(* IEC 61131-3 sources: AXOpen/src/components.rexroth.drives/app/src/IO, 9 files *)

(* ---- HwIdentifiers.st ---- *)
NAMESPACE AXOpen.Components.Rexroth.Drives
    TYPE
        HwIdentifiers : WORD
        (
            ST3_indradrive_HwID :=	WORD#258,
            ST3_indradrive_F_Modul_not_used_ID_FMod_NotUsed_HwID :=	WORD#266,
            ST3_indradrive_Input_9_Words_ID_InMod_9Words_HwID :=	WORD#264,
            ST3_indradrive_Output_13_Words_ID_OutMod_13Words_HwID :=	WORD#263,
            ST3_indradrive_ParamCh_5Words_ID_PaCh_5Words_HwID :=	WORD#265,
            ST3_indradrive_Rack_HwID :=	WORD#261,
            ST3_indradrive_ST3_indradrive_HwID :=	WORD#262,
            ST3_indradrive_ST3_indradrive_DAP_1_HwID :=	WORD#267,
            ST3_indradrive_ST3_indradrive_profinet_HwID :=	WORD#257,
            ST3_indradrive_ST3_indradrive_profinet_Port_1_HwID :=	WORD#259,
            ST3_indradrive_ST3_indradrive_profinet_Port_2_HwID :=	WORD#260,
            plc_line_HwID :=	WORD#32,
            plc_line_Rail_0_HwID :=	WORD#268,
            plc_line_plc_line_HwID :=	WORD#48,
            plc_line_plc_line_CPU_display_1_HwID :=	WORD#54,
            plc_line_plc_line_Card_reader_writer_1_HwID :=	WORD#51,
            plc_line_plc_line_DP_interface_1_HwID :=	WORD#60,
            plc_line_plc_line_OPC_UA_1_HwID :=	WORD#117,
            plc_line_plc_line_profinet_x1_HwID :=	WORD#64,
            plc_line_plc_line_profinet_x1_Port_1_HwID :=	WORD#65,
            plc_line_plc_line_profinet_x1_Port_2_HwID :=	WORD#66,
            plc_line_plc_line_profinet_x2_HwID :=	WORD#72,
            plc_line_plc_line_profinet_x2_Port_3_HwID :=	WORD#73,
            plc_line_plc_line_virtual_communication_interface_HwID :=	WORD#135,
            profinet_plc_line_HwID :=	WORD#256,

            NONE := WORD#0
        );
    END_TYPE
END_NAMESPACE

(* ---- HwInputs.st ---- *)
TYPE
	{S7.extern=ReadWrite}
	HwInputs : STRUCT
		ST3_indradrive_ParamCh_IDN_1 AT %B10 : ARRAY[0..9] OF BYTE;
		ST3_indradrive_Input_9_Words_1 AT %B20 : ARRAY[0..17] OF BYTE;
	END_STRUCT;
END_TYPE

(* ---- HwOutputs.st ---- *)
TYPE
	HwOutputs : STRUCT
		ST3_indradrive_ParamCh_IDN_1 AT %B10 : ARRAY[0..9] OF BYTE;
		ST3_indradrive_Output_13_Words_1 AT %B20 : ARRAY[0..25] OF BYTE;
	END_STRUCT;
END_TYPE

(* ---- Inputs.st ---- *)
NAMESPACE AXOpen.Components.Rexroth.Drives
    TYPE
        {S7.extern=ReadWrite}
        {#ix-attr:[Container(Layout.Wrap)]}
        Inputs : STRUCT
            AxoCtrlxDriveXsc_Inputs_Submodule_1 AT %B0:  WORD;
            AxoCtrlxDriveXsc_Inputs_Submodule_2 AT %B20:  WORD;
            AxoCtrlxDriveXsc_Inputs_Submodule_3 AT %B18:  WORD;
            AxoCtrlxDriveXsc_Inputs_Submodule_4 AT %B2:  WORD;
            AxoCtrlxDriveXsc_Inputs_Submodule_5 AT %B4:  DWORD;
            AxoCtrlxDriveXsc_Inputs_Submodule_6 AT %B12:  DWORD;
            AxoCtrlxDriveXsc_Inputs_Submodule_7 AT %B8:  DWORD;
            AxoCtrlxDriveXsc_Inputs_Submodule_8 AT %B16:  WORD;
            ST3_indradrive_Input_9_Words_0 AT %B24:  WORD;
            ST3_indradrive_Input_9_Words_1 AT %B26:  WORD;
            ST3_indradrive_Input_9_Words_2 AT %B28:  WORD;
            ST3_indradrive_Input_9_Words_3 AT %B30:  WORD;
            ST3_indradrive_Input_9_Words_4 AT %B32:  WORD;
            ST3_indradrive_Input_9_Words_5 AT %B34:  WORD;
            ST3_indradrive_Input_9_Words_6 AT %B36:  WORD;
            ST3_indradrive_Input_9_Words_7 AT %B38:  WORD;
            ST3_indradrive_Input_9_Words_8 AT %B40:  WORD;
            ST3_indradrive_ParamCh_5Words_0 AT %B42:  WORD;
            ST3_indradrive_ParamCh_5Words_1 AT %B44:  WORD;
            ST3_indradrive_ParamCh_5Words_2 AT %B46:  WORD;
            ST3_indradrive_ParamCh_5Words_3 AT %B48:  WORD;
            ST3_indradrive_ParamCh_5Words_4 AT %B50:  WORD;
        END_STRUCT;
    END_TYPE
END_NAMESPACE

(* ---- IoStructures.st ---- *)
NAMESPACE AXOpen.Components.Rexroth.Drives
	TYPE
        {S7.extern=ReadWrite}
        {#ix-attr:[Container(Layout.Wrap)]}
	    AxoCtrlxDriveXsc_Inputs_P_0_0106_0_0__STO_function__Operating_status_Input_Layout : STRUCT
	        Signals_0 AT %B0 : WORD;
	    END_STRUCT;
	END_TYPE

	TYPE
        {S7.extern=ReadWrite}
        {#ix-attr:[Container(Layout.Wrap)]}
	    AxoCtrlxDriveXsc_Inputs_S_0_0084_0_0__Torque_force_feedback_value_Input_Layout : STRUCT
	        Signals_0 AT %B0 : INT;
	    END_STRUCT;
	END_TYPE

	TYPE
        {S7.extern=ReadWrite}
        {#ix-attr:[Container(Layout.Wrap)]}
	    AxoCtrlxDriveXsc_Inputs_S_0_0135_0_0__Drive_status_word__Value_Input_Layout : STRUCT
	        Signals_0 AT %X0.3 : BOOL;
	        Signals_1 AT %X0.4 : BOOL;
	        Signals_2 AT %X0.5 : BOOL;
	        Signals_3 AT %X0.7 : BOOL;
	        Signals_4 AT %X1.0 : BOOL;
	        Signals_5 AT %X1.1 : BOOL;
	        Signals_6 AT %X1.2 : BOOL;
	        Signals_7 AT %X1.4 : BOOL;
	        Signals_8 AT %X1.5 : BOOL;
	        Signals_9 AT %X1.6 : BOOL;
	        Signals_10 AT %X1.7 : BOOL;
	    END_STRUCT;
	END_TYPE

	TYPE
        {S7.extern=ReadWrite}
        {#ix-attr:[Container(Layout.Wrap)]}
	    AxoCtrlxDriveXsc_Inputs_S_0_0144_0_0__Signal_status_word__Value_Input_Layout : STRUCT
	        Signals_0 AT %B0 : WORD;
	    END_STRUCT;
	END_TYPE

	TYPE
        {S7.extern=ReadWrite}
        {#ix-attr:[Container(Layout.Wrap)]}
	    AxoCtrlxDriveXsc_Inputs_S_0_0386_0_0__Position_controller__Position_actual_value_Input_Layout : STRUCT
	        Signals_0 AT %B0 : DINT;
	    END_STRUCT;
	END_TYPE

	TYPE
        {S7.extern=ReadWrite}
        {#ix-attr:[Container(Layout.Wrap)]}
	    AxoCtrlxDriveXsc_Inputs_S_0_0390_0_0__Diagnostic_message__Manufacturer_status_register_Input_Layout : STRUCT
	        Signals_0 AT %B0 : DWORD;
	    END_STRUCT;
	END_TYPE

	TYPE
        {S7.extern=ReadWrite}
        {#ix-attr:[Container(Layout.Wrap)]}
	    AxoCtrlxDriveXsc_Inputs_S_0_0535_0_0__Velocity_controller__Velocity_actual_value_Input_Layout : STRUCT
	        Signals_0 AT %B0 : DINT;
	    END_STRUCT;
	END_TYPE

	TYPE
        {S7.extern=ReadWrite}
        {#ix-attr:[Container(Layout.Wrap)]}
	    AxoCtrlxDriveXsc_Inputs_S_0_1720_0_2__Power_supply_control__Status_word_Input_Layout : STRUCT
	        Signals_0 AT %B0 : WORD;
	    END_STRUCT;
	END_TYPE

	TYPE
        {S7.extern=ReadWrite}
        {#ix-attr:[Container(Layout.Wrap)]}
	    AxoCtrlxDriveXsc_Outputs_S_0_0080_0_0__Torque_force_command_value_Output_Layout : STRUCT
	        Signals_0 AT %B0 : INT;
	    END_STRUCT;
	END_TYPE

	TYPE
        {S7.extern=ReadWrite}
        {#ix-attr:[Container(Layout.Wrap)]}
	    AxoCtrlxDriveXsc_Outputs_S_0_0092_0_0__Torque_force_limitation__Limit_value_bipolar_Output_Layout : STRUCT
	        Signals_0 AT %B0 : WORD;
	    END_STRUCT;
	END_TYPE

	TYPE
        {S7.extern=ReadWrite}
        {#ix-attr:[Container(Layout.Wrap)]}
	    AxoCtrlxDriveXsc_Outputs_S_0_0134_0_0__Master_control_word__Value_Output_Layout : STRUCT
	        Signals_0 AT %X1.0 : BOOL;
	        Signals_1 AT %X1.1 : BOOL;
	        Signals_2 AT %X1.2 : BOOL;
	        Signals_3 AT %X1.5 : BOOL;
	        Signals_4 AT %X1.6 : BOOL;
	        Signals_5 AT %X1.7 : BOOL;
	    END_STRUCT;
	END_TYPE

	TYPE
        {S7.extern=ReadWrite}
        {#ix-attr:[Container(Layout.Wrap)]}
	    AxoCtrlxDriveXsc_Outputs_S_0_0145_0_0__Signal_control_word__Value_Output_Layout : STRUCT
	        Signals_0 AT %B0 : WORD;
	    END_STRUCT;
	END_TYPE

	TYPE
        {S7.extern=ReadWrite}
        {#ix-attr:[Container(Layout.Wrap)]}
	    AxoCtrlxDriveXsc_Outputs_S_0_0193_0_0__Positioning_jerk_Output_Layout : STRUCT
	        Signals_0 AT %B0 : DINT;
	    END_STRUCT;
	END_TYPE

	TYPE
        {S7.extern=ReadWrite}
        {#ix-attr:[Container(Layout.Wrap)]}
	    AxoCtrlxDriveXsc_Outputs_S_0_0259_0_0__Positioning_profile__Profile_velocity_Output_Layout : STRUCT
	        Signals_0 AT %B0 : DWORD;
	    END_STRUCT;
	END_TYPE

	TYPE
        {S7.extern=ReadWrite}
        {#ix-attr:[Container(Layout.Wrap)]}
	    AxoCtrlxDriveXsc_Outputs_S_0_0260_0_0__Positioning_profile__Acceleration_Output_Layout : STRUCT
	        Signals_0 AT %B0 : DINT;
	    END_STRUCT;
	END_TYPE

	TYPE
        {S7.extern=ReadWrite}
        {#ix-attr:[Container(Layout.Wrap)]}
	    AxoCtrlxDriveXsc_Outputs_S_0_0282_0_0__Drive_controlled_positioning__Command_value_Output_Layout : STRUCT
	        Signals_0 AT %B0 : DINT;
	    END_STRUCT;
	END_TYPE

	TYPE
        {S7.extern=ReadWrite}
        {#ix-attr:[Container(Layout.Wrap)]}
	    AxoCtrlxDriveXsc_Outputs_S_0_0359_0_0__Positioning_profile__Deceleration_Output_Layout : STRUCT
	        Signals_0 AT %B0 : DINT;
	    END_STRUCT;
	END_TYPE

	TYPE
        {S7.extern=ReadWrite}
        {#ix-attr:[Container(Layout.Wrap)]}
	    AxoCtrlxDriveXsc_Outputs_S_0_1720_0_1__Power_supply_control__Control_word_Output_Layout : STRUCT
	        Signals_0 AT %B0 : WORD;
	    END_STRUCT;
	END_TYPE

	TYPE
        {S7.extern=ReadWrite}
        {#ix-attr:[Container(Layout.Wrap)]}
	    ST3_indradrive_Input_9_Words_Input_Layout : STRUCT
	        Signals_0 AT %B0 : WORD;
	        Signals_1 AT %B2 : WORD;
	        Signals_2 AT %B4 : WORD;
	        Signals_3 AT %B6 : WORD;
	        Signals_4 AT %B8 : WORD;
	        Signals_5 AT %B10 : WORD;
	        Signals_6 AT %B12 : WORD;
	        Signals_7 AT %B14 : WORD;
	        Signals_8 AT %B16 : WORD;
	    END_STRUCT;
	END_TYPE

	TYPE
        {S7.extern=ReadWrite}
        {#ix-attr:[Container(Layout.Wrap)]}
	    ST3_indradrive_Output_13_Words_Output_Layout : STRUCT
	        Signals_0 AT %B0 : WORD;
	        Signals_1 AT %B2 : WORD;
	        Signals_2 AT %B4 : WORD;
	        Signals_3 AT %B6 : WORD;
	        Signals_4 AT %B8 : WORD;
	        Signals_5 AT %B10 : WORD;
	        Signals_6 AT %B12 : WORD;
	        Signals_7 AT %B14 : WORD;
	        Signals_8 AT %B16 : WORD;
	        Signals_9 AT %B18 : WORD;
	        Signals_10 AT %B20 : WORD;
	        Signals_11 AT %B22 : WORD;
	        Signals_12 AT %B24 : WORD;
	    END_STRUCT;
	END_TYPE

	TYPE
        {S7.extern=ReadWrite}
        {#ix-attr:[Container(Layout.Wrap)]}
	    ST3_indradrive_ParamCh_5Words_Input_Layout : STRUCT
	        Signals_0 AT %B0 : WORD;
	        Signals_1 AT %B2 : WORD;
	        Signals_2 AT %B4 : WORD;
	        Signals_3 AT %B6 : WORD;
	        Signals_4 AT %B8 : WORD;
	    END_STRUCT;
	END_TYPE

	TYPE
        {S7.extern=ReadWrite}
        {#ix-attr:[Container(Layout.Wrap)]}
	    ST3_indradrive_ParamCh_5Words_Output_Layout : STRUCT
	        Signals_5 AT %B0 : WORD;
	        Signals_6 AT %B2 : WORD;
	        Signals_7 AT %B4 : WORD;
	        Signals_8 AT %B6 : WORD;
	        Signals_9 AT %B8 : WORD;
	    END_STRUCT;
	END_TYPE
END_NAMESPACE

(* ---- Outputs.st ---- *)
NAMESPACE AXOpen.Components.Rexroth.Drives
    TYPE
        {S7.extern=ReadWrite}
        {#ix-attr:[Container(Layout.Wrap)]}
        Outputs : STRUCT
	        // Module rexroth_ctrlx_drive/Outputs
	        rexroth_ctrlx_drive_Outputs_S_0_0080_0_0__Torque_force_command_value_Output AT %B24 : rexroth_ctrlx_drive_Outputs_S_0_0080_0_0__Torque_force_command_value_Output_Layout;

	        rexroth_ctrlx_drive_Outputs_S_0_0092_0_0__Torque_force_limitation__Limit_value_bipolar_Output AT %B22 : rexroth_ctrlx_drive_Outputs_S_0_0092_0_0__Torque_force_limitation__Limit_value_bipolar_Output_Layout;

	        rexroth_ctrlx_drive_Outputs_S_0_0134_0_0__Master_control_word__Value_Output AT %B0 : rexroth_ctrlx_drive_Outputs_S_0_0134_0_0__Master_control_word__Value_Output_Layout;

	        rexroth_ctrlx_drive_Outputs_S_0_0145_0_0__Signal_control_word__Value_Output AT %B18 : rexroth_ctrlx_drive_Outputs_S_0_0145_0_0__Signal_control_word__Value_Output_Layout;

	        rexroth_ctrlx_drive_Outputs_S_0_0193_0_0__Positioning_jerk_Output AT %B26 : rexroth_ctrlx_drive_Outputs_S_0_0193_0_0__Positioning_jerk_Output_Layout;

	        rexroth_ctrlx_drive_Outputs_S_0_0259_0_0__Positioning_profile__Profile_velocity_Output AT %B14 : rexroth_ctrlx_drive_Outputs_S_0_0259_0_0__Positioning_profile__Profile_velocity_Output_Layout;

	        rexroth_ctrlx_drive_Outputs_S_0_0260_0_0__Positioning_profile__Acceleration_Output AT %B2 : rexroth_ctrlx_drive_Outputs_S_0_0260_0_0__Positioning_profile__Acceleration_Output_Layout;

	        rexroth_ctrlx_drive_Outputs_S_0_0282_0_0__Drive_controlled_positioning__Command_value_Output AT %B6 : rexroth_ctrlx_drive_Outputs_S_0_0282_0_0__Drive_controlled_positioning__Command_value_Output_Layout;

	        rexroth_ctrlx_drive_Outputs_S_0_0359_0_0__Positioning_profile__Deceleration_Output AT %B10 : rexroth_ctrlx_drive_Outputs_S_0_0359_0_0__Positioning_profile__Deceleration_Output_Layout;

	        rexroth_ctrlx_drive_Outputs_S_0_1720_0_1__Power_supply_control__Control_word_Output AT %B20 : rexroth_ctrlx_drive_Outputs_S_0_1720_0_1__Power_supply_control__Control_word_Output_Layout;

	        // Module rexroth_indradrive/Output_13_Words
	        rexroth_indradrive_Output_13_Words_Output AT %B30 : rexroth_indradrive_Output_13_Words_Output_Layout;

	        rexroth_indradrive_ParamCh_5Words_Output AT %B56 : rexroth_indradrive_ParamCh_5Words_Output_Layout;

        END_STRUCT;
    END_TYPE
END_NAMESPACE

(* ---- PlcInputs.st ---- *)
TYPE
	PlcInputs : STRUCT
		ST3_indradrive_ParamCh_IDN_1 : ARRAY[0..9] OF BYTE;
		ST3_indradrive_Input_9_Words_1 : ARRAY[0..17] OF BYTE;
	END_STRUCT;
END_TYPE

(* ---- PlcOutputs.st ---- *)
TYPE
	PlcOutputs : STRUCT
		ST3_indradrive_ParamCh_IDN_1 : ARRAY[0..9] OF BYTE;
		ST3_indradrive_Output_13_Words_1 : ARRAY[0..25] OF BYTE;
	END_STRUCT;
END_TYPE

(* ---- CopyInputs.st ---- *)
FUNCTION CopyInputs
	VAR_EXTERNAL
		HwInputs : HwInputs;
		PlcInputs : PlcInputs;
	END_VAR
	PlcInputs._10a1_Acquisition_Status_1[0] := HwInputs._10a1_Acquisition_Status_1[0];
	PlcInputs._10a1_Acquisition_Status_1[1] := HwInputs._10a1_Acquisition_Status_1[1];
	PlcInputs._10a1_Acquisition_Status_1[2] := HwInputs._10a1_Acquisition_Status_1[2];
	PlcInputs._10a1_Results_Status_1 := HwInputs._10a1_Results_Status_1;
	PlcInputs._10a1_Soft_Event_Control_1 := HwInputs._10a1_Soft_Event_Control_1;
	PlcInputs._10a1_Result_Data_128_bytes_1[0] := HwInputs._10a1_Result_Data_128_bytes_1[0];
	PlcInputs._10a1_Result_Data_128_bytes_1[1] := HwInputs._10a1_Result_Data_128_bytes_1[1];
	PlcInputs._10a1_Result_Data_128_bytes_1[2] := HwInputs._10a1_Result_Data_128_bytes_1[2];
	PlcInputs._10a1_Result_Data_128_bytes_1[3] := HwInputs._10a1_Result_Data_128_bytes_1[3];
	PlcInputs._10a1_Result_Data_128_bytes_1[4] := HwInputs._10a1_Result_Data_128_bytes_1[4];
	PlcInputs._10a1_Result_Data_128_bytes_1[5] := HwInputs._10a1_Result_Data_128_bytes_1[5];
	PlcInputs._10a1_Result_Data_128_bytes_1[6] := HwInputs._10a1_Result_Data_128_bytes_1[6];
	PlcInputs._10a1_Result_Data_128_bytes_1[7] := HwInputs._10a1_Result_Data_128_bytes_1[7];
	PlcInputs._10a1_Result_Data_128_bytes_1[8] := HwInputs._10a1_Result_Data_128_bytes_1[8];
	PlcInputs._10a1_Result_Data_128_bytes_1[9] := HwInputs._10a1_Result_Data_128_bytes_1[9];
	PlcInputs._10a1_Result_Data_128_bytes_1[10] := HwInputs._10a1_Result_Data_128_bytes_1[10];
	PlcInputs._10a1_Result_Data_128_bytes_1[11] := HwInputs._10a1_Result_Data_128_bytes_1[11];
	PlcInputs._10a1_Result_Data_128_bytes_1[12] := HwInputs._10a1_Result_Data_128_bytes_1[12];
	PlcInputs._10a1_Result_Data_128_bytes_1[13] := HwInputs._10a1_Result_Data_128_bytes_1[13];
	PlcInputs._10a1_Result_Data_128_bytes_1[14] := HwInputs._10a1_Result_Data_128_bytes_1[14];
	PlcInputs._10a1_Result_Data_128_bytes_1[15] := HwInputs._10a1_Result_Data_128_bytes_1[15];
	PlcInputs._10a1_Result_Data_128_bytes_1[16] := HwInputs._10a1_Result_Data_128_bytes_1[16];
	PlcInputs._10a1_Result_Data_128_bytes_1[17] := HwInputs._10a1_Result_Data_128_bytes_1[17];
	PlcInputs._10a1_Result_Data_128_bytes_1[18] := HwInputs._10a1_Result_Data_128_bytes_1[18];
	PlcInputs._10a1_Result_Data_128_bytes_1[19] := HwInputs._10a1_Result_Data_128_bytes_1[19];
	PlcInputs._10a1_Result_Data_128_bytes_1[20] := HwInputs._10a1_Result_Data_128_bytes_1[20];
	PlcInputs._10a1_Result_Data_128_bytes_1[21] := HwInputs._10a1_Result_Data_128_bytes_1[21];
	PlcInputs._10a1_Result_Data_128_bytes_1[22] := HwInputs._10a1_Result_Data_128_bytes_1[22];
	PlcInputs._10a1_Result_Data_128_bytes_1[23] := HwInputs._10a1_Result_Data_128_bytes_1[23];
	PlcInputs._10a1_Result_Data_128_bytes_1[24] := HwInputs._10a1_Result_Data_128_bytes_1[24];
	PlcInputs._10a1_Result_Data_128_bytes_1[25] := HwInputs._10a1_Result_Data_128_bytes_1[25];
	PlcInputs._10a1_Result_Data_128_bytes_1[26] := HwInputs._10a1_Result_Data_128_bytes_1[26];
	PlcInputs._10a1_Result_Data_128_bytes_1[27] := HwInputs._10a1_Result_Data_128_bytes_1[27];
	PlcInputs._10a1_Result_Data_128_bytes_1[28] := HwInputs._10a1_Result_Data_128_bytes_1[28];
	PlcInputs._10a1_Result_Data_128_bytes_1[29] := HwInputs._10a1_Result_Data_128_bytes_1[29];
	PlcInputs._10a1_Result_Data_128_bytes_1[30] := HwInputs._10a1_Result_Data_128_bytes_1[30];
	PlcInputs._10a1_Result_Data_128_bytes_1[31] := HwInputs._10a1_Result_Data_128_bytes_1[31];
	PlcInputs._10a1_Result_Data_128_bytes_1[32] := HwInputs._10a1_Result_Data_128_bytes_1[32];
	PlcInputs._10a1_Result_Data_128_bytes_1[33] := HwInputs._10a1_Result_Data_128_bytes_1[33];
	PlcInputs._10a1_Result_Data_128_bytes_1[34] := HwInputs._10a1_Result_Data_128_bytes_1[34];
	PlcInputs._10a1_Result_Data_128_bytes_1[35] := HwInputs._10a1_Result_Data_128_bytes_1[35];
	PlcInputs._10a1_Result_Data_128_bytes_1[36] := HwInputs._10a1_Result_Data_128_bytes_1[36];
	PlcInputs._10a1_Result_Data_128_bytes_1[37] := HwInputs._10a1_Result_Data_128_bytes_1[37];
	PlcInputs._10a1_Result_Data_128_bytes_1[38] := HwInputs._10a1_Result_Data_128_bytes_1[38];
	PlcInputs._10a1_Result_Data_128_bytes_1[39] := HwInputs._10a1_Result_Data_128_bytes_1[39];
	PlcInputs._10a1_Result_Data_128_bytes_1[40] := HwInputs._10a1_Result_Data_128_bytes_1[40];
	PlcInputs._10a1_Result_Data_128_bytes_1[41] := HwInputs._10a1_Result_Data_128_bytes_1[41];
	PlcInputs._10a1_Result_Data_128_bytes_1[42] := HwInputs._10a1_Result_Data_128_bytes_1[42];
	PlcInputs._10a1_Result_Data_128_bytes_1[43] := HwInputs._10a1_Result_Data_128_bytes_1[43];
	PlcInputs._10a1_Result_Data_128_bytes_1[44] := HwInputs._10a1_Result_Data_128_bytes_1[44];
	PlcInputs._10a1_Result_Data_128_bytes_1[45] := HwInputs._10a1_Result_Data_128_bytes_1[45];
	PlcInputs._10a1_Result_Data_128_bytes_1[46] := HwInputs._10a1_Result_Data_128_bytes_1[46];
	PlcInputs._10a1_Result_Data_128_bytes_1[47] := HwInputs._10a1_Result_Data_128_bytes_1[47];
	PlcInputs._10a1_Result_Data_128_bytes_1[48] := HwInputs._10a1_Result_Data_128_bytes_1[48];
	PlcInputs._10a1_Result_Data_128_bytes_1[49] := HwInputs._10a1_Result_Data_128_bytes_1[49];
	PlcInputs._10a1_Result_Data_128_bytes_1[50] := HwInputs._10a1_Result_Data_128_bytes_1[50];
	PlcInputs._10a1_Result_Data_128_bytes_1[51] := HwInputs._10a1_Result_Data_128_bytes_1[51];
	PlcInputs._10a1_Result_Data_128_bytes_1[52] := HwInputs._10a1_Result_Data_128_bytes_1[52];
	PlcInputs._10a1_Result_Data_128_bytes_1[53] := HwInputs._10a1_Result_Data_128_bytes_1[53];
	PlcInputs._10a1_Result_Data_128_bytes_1[54] := HwInputs._10a1_Result_Data_128_bytes_1[54];
	PlcInputs._10a1_Result_Data_128_bytes_1[55] := HwInputs._10a1_Result_Data_128_bytes_1[55];
	PlcInputs._10a1_Result_Data_128_bytes_1[56] := HwInputs._10a1_Result_Data_128_bytes_1[56];
	PlcInputs._10a1_Result_Data_128_bytes_1[57] := HwInputs._10a1_Result_Data_128_bytes_1[57];
	PlcInputs._10a1_Result_Data_128_bytes_1[58] := HwInputs._10a1_Result_Data_128_bytes_1[58];
	PlcInputs._10a1_Result_Data_128_bytes_1[59] := HwInputs._10a1_Result_Data_128_bytes_1[59];
	PlcInputs._10a1_Result_Data_128_bytes_1[60] := HwInputs._10a1_Result_Data_128_bytes_1[60];
	PlcInputs._10a1_Result_Data_128_bytes_1[61] := HwInputs._10a1_Result_Data_128_bytes_1[61];
	PlcInputs._10a1_Result_Data_128_bytes_1[62] := HwInputs._10a1_Result_Data_128_bytes_1[62];
	PlcInputs._10a1_Result_Data_128_bytes_1[63] := HwInputs._10a1_Result_Data_128_bytes_1[63];
	PlcInputs._10a1_Result_Data_128_bytes_1[64] := HwInputs._10a1_Result_Data_128_bytes_1[64];
	PlcInputs._10a1_Result_Data_128_bytes_1[65] := HwInputs._10a1_Result_Data_128_bytes_1[65];
	PlcInputs._10a1_Result_Data_128_bytes_1[66] := HwInputs._10a1_Result_Data_128_bytes_1[66];
	PlcInputs._10a1_Result_Data_128_bytes_1[67] := HwInputs._10a1_Result_Data_128_bytes_1[67];
	PlcInputs._10a1_Result_Data_128_bytes_1[68] := HwInputs._10a1_Result_Data_128_bytes_1[68];
	PlcInputs._10a1_Result_Data_128_bytes_1[69] := HwInputs._10a1_Result_Data_128_bytes_1[69];
	PlcInputs._10a1_Result_Data_128_bytes_1[70] := HwInputs._10a1_Result_Data_128_bytes_1[70];
	PlcInputs._10a1_Result_Data_128_bytes_1[71] := HwInputs._10a1_Result_Data_128_bytes_1[71];
	PlcInputs._10a1_Result_Data_128_bytes_1[72] := HwInputs._10a1_Result_Data_128_bytes_1[72];
	PlcInputs._10a1_Result_Data_128_bytes_1[73] := HwInputs._10a1_Result_Data_128_bytes_1[73];
	PlcInputs._10a1_Result_Data_128_bytes_1[74] := HwInputs._10a1_Result_Data_128_bytes_1[74];
	PlcInputs._10a1_Result_Data_128_bytes_1[75] := HwInputs._10a1_Result_Data_128_bytes_1[75];
	PlcInputs._10a1_Result_Data_128_bytes_1[76] := HwInputs._10a1_Result_Data_128_bytes_1[76];
	PlcInputs._10a1_Result_Data_128_bytes_1[77] := HwInputs._10a1_Result_Data_128_bytes_1[77];
	PlcInputs._10a1_Result_Data_128_bytes_1[78] := HwInputs._10a1_Result_Data_128_bytes_1[78];
	PlcInputs._10a1_Result_Data_128_bytes_1[79] := HwInputs._10a1_Result_Data_128_bytes_1[79];
	PlcInputs._10a1_Result_Data_128_bytes_1[80] := HwInputs._10a1_Result_Data_128_bytes_1[80];
	PlcInputs._10a1_Result_Data_128_bytes_1[81] := HwInputs._10a1_Result_Data_128_bytes_1[81];
	PlcInputs._10a1_Result_Data_128_bytes_1[82] := HwInputs._10a1_Result_Data_128_bytes_1[82];
	PlcInputs._10a1_Result_Data_128_bytes_1[83] := HwInputs._10a1_Result_Data_128_bytes_1[83];
	PlcInputs._10a1_Result_Data_128_bytes_1[84] := HwInputs._10a1_Result_Data_128_bytes_1[84];
	PlcInputs._10a1_Result_Data_128_bytes_1[85] := HwInputs._10a1_Result_Data_128_bytes_1[85];
	PlcInputs._10a1_Result_Data_128_bytes_1[86] := HwInputs._10a1_Result_Data_128_bytes_1[86];
	PlcInputs._10a1_Result_Data_128_bytes_1[87] := HwInputs._10a1_Result_Data_128_bytes_1[87];
	PlcInputs._10a1_Result_Data_128_bytes_1[88] := HwInputs._10a1_Result_Data_128_bytes_1[88];
	PlcInputs._10a1_Result_Data_128_bytes_1[89] := HwInputs._10a1_Result_Data_128_bytes_1[89];
	PlcInputs._10a1_Result_Data_128_bytes_1[90] := HwInputs._10a1_Result_Data_128_bytes_1[90];
	PlcInputs._10a1_Result_Data_128_bytes_1[91] := HwInputs._10a1_Result_Data_128_bytes_1[91];
	PlcInputs._10a1_Result_Data_128_bytes_1[92] := HwInputs._10a1_Result_Data_128_bytes_1[92];
	PlcInputs._10a1_Result_Data_128_bytes_1[93] := HwInputs._10a1_Result_Data_128_bytes_1[93];
	PlcInputs._10a1_Result_Data_128_bytes_1[94] := HwInputs._10a1_Result_Data_128_bytes_1[94];
	PlcInputs._10a1_Result_Data_128_bytes_1[95] := HwInputs._10a1_Result_Data_128_bytes_1[95];
	PlcInputs._10a1_Result_Data_128_bytes_1[96] := HwInputs._10a1_Result_Data_128_bytes_1[96];
	PlcInputs._10a1_Result_Data_128_bytes_1[97] := HwInputs._10a1_Result_Data_128_bytes_1[97];
	PlcInputs._10a1_Result_Data_128_bytes_1[98] := HwInputs._10a1_Result_Data_128_bytes_1[98];
	PlcInputs._10a1_Result_Data_128_bytes_1[99] := HwInputs._10a1_Result_Data_128_bytes_1[99];
	PlcInputs._10a1_Result_Data_128_bytes_1[100] := HwInputs._10a1_Result_Data_128_bytes_1[100];
	PlcInputs._10a1_Result_Data_128_bytes_1[101] := HwInputs._10a1_Result_Data_128_bytes_1[101];
	PlcInputs._10a1_Result_Data_128_bytes_1[102] := HwInputs._10a1_Result_Data_128_bytes_1[102];
	PlcInputs._10a1_Result_Data_128_bytes_1[103] := HwInputs._10a1_Result_Data_128_bytes_1[103];
	PlcInputs._10a1_Result_Data_128_bytes_1[104] := HwInputs._10a1_Result_Data_128_bytes_1[104];
	PlcInputs._10a1_Result_Data_128_bytes_1[105] := HwInputs._10a1_Result_Data_128_bytes_1[105];
	PlcInputs._10a1_Result_Data_128_bytes_1[106] := HwInputs._10a1_Result_Data_128_bytes_1[106];
	PlcInputs._10a1_Result_Data_128_bytes_1[107] := HwInputs._10a1_Result_Data_128_bytes_1[107];
	PlcInputs._10a1_Result_Data_128_bytes_1[108] := HwInputs._10a1_Result_Data_128_bytes_1[108];
	PlcInputs._10a1_Result_Data_128_bytes_1[109] := HwInputs._10a1_Result_Data_128_bytes_1[109];
	PlcInputs._10a1_Result_Data_128_bytes_1[110] := HwInputs._10a1_Result_Data_128_bytes_1[110];
	PlcInputs._10a1_Result_Data_128_bytes_1[111] := HwInputs._10a1_Result_Data_128_bytes_1[111];
	PlcInputs._10a1_Result_Data_128_bytes_1[112] := HwInputs._10a1_Result_Data_128_bytes_1[112];
	PlcInputs._10a1_Result_Data_128_bytes_1[113] := HwInputs._10a1_Result_Data_128_bytes_1[113];
	PlcInputs._10a1_Result_Data_128_bytes_1[114] := HwInputs._10a1_Result_Data_128_bytes_1[114];
	PlcInputs._10a1_Result_Data_128_bytes_1[115] := HwInputs._10a1_Result_Data_128_bytes_1[115];
	PlcInputs._10a1_Result_Data_128_bytes_1[116] := HwInputs._10a1_Result_Data_128_bytes_1[116];
	PlcInputs._10a1_Result_Data_128_bytes_1[117] := HwInputs._10a1_Result_Data_128_bytes_1[117];
	PlcInputs._10a1_Result_Data_128_bytes_1[118] := HwInputs._10a1_Result_Data_128_bytes_1[118];
	PlcInputs._10a1_Result_Data_128_bytes_1[119] := HwInputs._10a1_Result_Data_128_bytes_1[119];
	PlcInputs._10a1_Result_Data_128_bytes_1[120] := HwInputs._10a1_Result_Data_128_bytes_1[120];
	PlcInputs._10a1_Result_Data_128_bytes_1[121] := HwInputs._10a1_Result_Data_128_bytes_1[121];
	PlcInputs._10a1_Result_Data_128_bytes_1[122] := HwInputs._10a1_Result_Data_128_bytes_1[122];
	PlcInputs._10a1_Result_Data_128_bytes_1[123] := HwInputs._10a1_Result_Data_128_bytes_1[123];
	PlcInputs._10a1_Result_Data_128_bytes_1[124] := HwInputs._10a1_Result_Data_128_bytes_1[124];
	PlcInputs._10a1_Result_Data_128_bytes_1[125] := HwInputs._10a1_Result_Data_128_bytes_1[125];
	PlcInputs._10a1_Result_Data_128_bytes_1[126] := HwInputs._10a1_Result_Data_128_bytes_1[126];
	PlcInputs._10a1_Result_Data_128_bytes_1[127] := HwInputs._10a1_Result_Data_128_bytes_1[127];
	PlcInputs._10a1_Result_Data_128_bytes_1[128] := HwInputs._10a1_Result_Data_128_bytes_1[128];
	PlcInputs._10a1_Result_Data_128_bytes_1[129] := HwInputs._10a1_Result_Data_128_bytes_1[129];
	PlcInputs._10a1_Result_Data_128_bytes_1[130] := HwInputs._10a1_Result_Data_128_bytes_1[130];
	PlcInputs._10a1_Result_Data_128_bytes_1[131] := HwInputs._10a1_Result_Data_128_bytes_1[131];
	PlcInputs._10a1_Result_Data_128_bytes_1[132] := HwInputs._10a1_Result_Data_128_bytes_1[132];
	PlcInputs._10a1_Result_Data_128_bytes_1[133] := HwInputs._10a1_Result_Data_128_bytes_1[133];
	PlcInputs._10a1_Result_Data_128_bytes_1[134] := HwInputs._10a1_Result_Data_128_bytes_1[134];
	PlcInputs._10a1_Result_Data_128_bytes_1[135] := HwInputs._10a1_Result_Data_128_bytes_1[135];
	PlcInputs.reader_st2_Acquisition_Status_1[0] := HwInputs.reader_st2_Acquisition_Status_1[0];
	PlcInputs.reader_st2_Acquisition_Status_1[1] := HwInputs.reader_st2_Acquisition_Status_1[1];
	PlcInputs.reader_st2_Acquisition_Status_1[2] := HwInputs.reader_st2_Acquisition_Status_1[2];
	PlcInputs.reader_st2_Results_Status_1 := HwInputs.reader_st2_Results_Status_1;
	PlcInputs.reader_st2_Soft_Event_Control_1 := HwInputs.reader_st2_Soft_Event_Control_1;
	PlcInputs.reader_st2_Result_Data_64_bytes_1[0] := HwInputs.reader_st2_Result_Data_64_bytes_1[0];
	PlcInputs.reader_st2_Result_Data_64_bytes_1[1] := HwInputs.reader_st2_Result_Data_64_bytes_1[1];
	PlcInputs.reader_st2_Result_Data_64_bytes_1[2] := HwInputs.reader_st2_Result_Data_64_bytes_1[2];
	PlcInputs.reader_st2_Result_Data_64_bytes_1[3] := HwInputs.reader_st2_Result_Data_64_bytes_1[3];
	PlcInputs.reader_st2_Result_Data_64_bytes_1[4] := HwInputs.reader_st2_Result_Data_64_bytes_1[4];
	PlcInputs.reader_st2_Result_Data_64_bytes_1[5] := HwInputs.reader_st2_Result_Data_64_bytes_1[5];
	PlcInputs.reader_st2_Result_Data_64_bytes_1[6] := HwInputs.reader_st2_Result_Data_64_bytes_1[6];
	PlcInputs.reader_st2_Result_Data_64_bytes_1[7] := HwInputs.reader_st2_Result_Data_64_bytes_1[7];
	PlcInputs.reader_st2_Result_Data_64_bytes_1[8] := HwInputs.reader_st2_Result_Data_64_bytes_1[8];
	PlcInputs.reader_st2_Result_Data_64_bytes_1[9] := HwInputs.reader_st2_Result_Data_64_bytes_1[9];
	PlcInputs.reader_st2_Result_Data_64_bytes_1[10] := HwInputs.reader_st2_Result_Data_64_bytes_1[10];
	PlcInputs.reader_st2_Result_Data_64_bytes_1[11] := HwInputs.reader_st2_Result_Data_64_bytes_1[11];
	PlcInputs.reader_st2_Result_Data_64_bytes_1[12] := HwInputs.reader_st2_Result_Data_64_bytes_1[12];
	PlcInputs.reader_st2_Result_Data_64_bytes_1[13] := HwInputs.reader_st2_Result_Data_64_bytes_1[13];
	PlcInputs.reader_st2_Result_Data_64_bytes_1[14] := HwInputs.reader_st2_Result_Data_64_bytes_1[14];
	PlcInputs.reader_st2_Result_Data_64_bytes_1[15] := HwInputs.reader_st2_Result_Data_64_bytes_1[15];
	PlcInputs.reader_st2_Result_Data_64_bytes_1[16] := HwInputs.reader_st2_Result_Data_64_bytes_1[16];
	PlcInputs.reader_st2_Result_Data_64_bytes_1[17] := HwInputs.reader_st2_Result_Data_64_bytes_1[17];
	PlcInputs.reader_st2_Result_Data_64_bytes_1[18] := HwInputs.reader_st2_Result_Data_64_bytes_1[18];
	PlcInputs.reader_st2_Result_Data_64_bytes_1[19] := HwInputs.reader_st2_Result_Data_64_bytes_1[19];
	PlcInputs.reader_st2_Result_Data_64_bytes_1[20] := HwInputs.reader_st2_Result_Data_64_bytes_1[20];
	PlcInputs.reader_st2_Result_Data_64_bytes_1[21] := HwInputs.reader_st2_Result_Data_64_bytes_1[21];
	PlcInputs.reader_st2_Result_Data_64_bytes_1[22] := HwInputs.reader_st2_Result_Data_64_bytes_1[22];
	PlcInputs.reader_st2_Result_Data_64_bytes_1[23] := HwInputs.reader_st2_Result_Data_64_bytes_1[23];
	PlcInputs.reader_st2_Result_Data_64_bytes_1[24] := HwInputs.reader_st2_Result_Data_64_bytes_1[24];
	PlcInputs.reader_st2_Result_Data_64_bytes_1[25] := HwInputs.reader_st2_Result_Data_64_bytes_1[25];
	PlcInputs.reader_st2_Result_Data_64_bytes_1[26] := HwInputs.reader_st2_Result_Data_64_bytes_1[26];
	PlcInputs.reader_st2_Result_Data_64_bytes_1[27] := HwInputs.reader_st2_Result_Data_64_bytes_1[27];
	PlcInputs.reader_st2_Result_Data_64_bytes_1[28] := HwInputs.reader_st2_Result_Data_64_bytes_1[28];
	PlcInputs.reader_st2_Result_Data_64_bytes_1[29] := HwInputs.reader_st2_Result_Data_64_bytes_1[29];
	PlcInputs.reader_st2_Result_Data_64_bytes_1[30] := HwInputs.reader_st2_Result_Data_64_bytes_1[30];
	PlcInputs.reader_st2_Result_Data_64_bytes_1[31] := HwInputs.reader_st2_Result_Data_64_bytes_1[31];
	PlcInputs.reader_st2_Result_Data_64_bytes_1[32] := HwInputs.reader_st2_Result_Data_64_bytes_1[32];
	PlcInputs.reader_st2_Result_Data_64_bytes_1[33] := HwInputs.reader_st2_Result_Data_64_bytes_1[33];
	PlcInputs.reader_st2_Result_Data_64_bytes_1[34] := HwInputs.reader_st2_Result_Data_64_bytes_1[34];
	PlcInputs.reader_st2_Result_Data_64_bytes_1[35] := HwInputs.reader_st2_Result_Data_64_bytes_1[35];
	PlcInputs.reader_st2_Result_Data_64_bytes_1[36] := HwInputs.reader_st2_Result_Data_64_bytes_1[36];
	PlcInputs.reader_st2_Result_Data_64_bytes_1[37] := HwInputs.reader_st2_Result_Data_64_bytes_1[37];
	PlcInputs.reader_st2_Result_Data_64_bytes_1[38] := HwInputs.reader_st2_Result_Data_64_bytes_1[38];
	PlcInputs.reader_st2_Result_Data_64_bytes_1[39] := HwInputs.reader_st2_Result_Data_64_bytes_1[39];
	PlcInputs.reader_st2_Result_Data_64_bytes_1[40] := HwInputs.reader_st2_Result_Data_64_bytes_1[40];
	PlcInputs.reader_st2_Result_Data_64_bytes_1[41] := HwInputs.reader_st2_Result_Data_64_bytes_1[41];
	PlcInputs.reader_st2_Result_Data_64_bytes_1[42] := HwInputs.reader_st2_Result_Data_64_bytes_1[42];
	PlcInputs.reader_st2_Result_Data_64_bytes_1[43] := HwInputs.reader_st2_Result_Data_64_bytes_1[43];
	PlcInputs.reader_st2_Result_Data_64_bytes_1[44] := HwInputs.reader_st2_Result_Data_64_bytes_1[44];
	PlcInputs.reader_st2_Result_Data_64_bytes_1[45] := HwInputs.reader_st2_Result_Data_64_bytes_1[45];
	PlcInputs.reader_st2_Result_Data_64_bytes_1[46] := HwInputs.reader_st2_Result_Data_64_bytes_1[46];
	PlcInputs.reader_st2_Result_Data_64_bytes_1[47] := HwInputs.reader_st2_Result_Data_64_bytes_1[47];
	PlcInputs.reader_st2_Result_Data_64_bytes_1[48] := HwInputs.reader_st2_Result_Data_64_bytes_1[48];
	PlcInputs.reader_st2_Result_Data_64_bytes_1[49] := HwInputs.reader_st2_Result_Data_64_bytes_1[49];
	PlcInputs.reader_st2_Result_Data_64_bytes_1[50] := HwInputs.reader_st2_Result_Data_64_bytes_1[50];
	PlcInputs.reader_st2_Result_Data_64_bytes_1[51] := HwInputs.reader_st2_Result_Data_64_bytes_1[51];
	PlcInputs.reader_st2_Result_Data_64_bytes_1[52] := HwInputs.reader_st2_Result_Data_64_bytes_1[52];
	PlcInputs.reader_st2_Result_Data_64_bytes_1[53] := HwInputs.reader_st2_Result_Data_64_bytes_1[53];
	PlcInputs.reader_st2_Result_Data_64_bytes_1[54] := HwInputs.reader_st2_Result_Data_64_bytes_1[54];
	PlcInputs.reader_st2_Result_Data_64_bytes_1[55] := HwInputs.reader_st2_Result_Data_64_bytes_1[55];
	PlcInputs.reader_st2_Result_Data_64_bytes_1[56] := HwInputs.reader_st2_Result_Data_64_bytes_1[56];
	PlcInputs.reader_st2_Result_Data_64_bytes_1[57] := HwInputs.reader_st2_Result_Data_64_bytes_1[57];
	PlcInputs.reader_st2_Result_Data_64_bytes_1[58] := HwInputs.reader_st2_Result_Data_64_bytes_1[58];
	PlcInputs.reader_st2_Result_Data_64_bytes_1[59] := HwInputs.reader_st2_Result_Data_64_bytes_1[59];
	PlcInputs.reader_st2_Result_Data_64_bytes_1[60] := HwInputs.reader_st2_Result_Data_64_bytes_1[60];
	PlcInputs.reader_st2_Result_Data_64_bytes_1[61] := HwInputs.reader_st2_Result_Data_64_bytes_1[61];
	PlcInputs.reader_st2_Result_Data_64_bytes_1[62] := HwInputs.reader_st2_Result_Data_64_bytes_1[62];
	PlcInputs.reader_st2_Result_Data_64_bytes_1[63] := HwInputs.reader_st2_Result_Data_64_bytes_1[63];
	PlcInputs.reader_st2_Result_Data_64_bytes_1[64] := HwInputs.reader_st2_Result_Data_64_bytes_1[64];
	PlcInputs.reader_st2_Result_Data_64_bytes_1[65] := HwInputs.reader_st2_Result_Data_64_bytes_1[65];
	PlcInputs.reader_st2_Result_Data_64_bytes_1[66] := HwInputs.reader_st2_Result_Data_64_bytes_1[66];
	PlcInputs.reader_st2_Result_Data_64_bytes_1[67] := HwInputs.reader_st2_Result_Data_64_bytes_1[67];
	PlcInputs.reader_st2_Result_Data_64_bytes_1[68] := HwInputs.reader_st2_Result_Data_64_bytes_1[68];
	PlcInputs.reader_st2_Result_Data_64_bytes_1[69] := HwInputs.reader_st2_Result_Data_64_bytes_1[69];
	PlcInputs.reader_st2_Result_Data_64_bytes_1[70] := HwInputs.reader_st2_Result_Data_64_bytes_1[70];
	PlcInputs.reader_st2_Result_Data_64_bytes_1[71] := HwInputs.reader_st2_Result_Data_64_bytes_1[71];
	PlcInputs._7600_Acquisition_Status_1[0] := HwInputs._7600_Acquisition_Status_1[0];
	PlcInputs._7600_Acquisition_Status_1[1] := HwInputs._7600_Acquisition_Status_1[1];
	PlcInputs._7600_Acquisition_Status_1[2] := HwInputs._7600_Acquisition_Status_1[2];
	PlcInputs._7600_Inspection_Status_1 := HwInputs._7600_Inspection_Status_1;
	PlcInputs._7600_Command_Control_1 := HwInputs._7600_Command_Control_1;
	PlcInputs._7600_SoftEvent_Control_1 := HwInputs._7600_SoftEvent_Control_1;
	PlcInputs._7600_Results_64_bytes_1[0] := HwInputs._7600_Results_64_bytes_1[0];
	PlcInputs._7600_Results_64_bytes_1[1] := HwInputs._7600_Results_64_bytes_1[1];
	PlcInputs._7600_Results_64_bytes_1[2] := HwInputs._7600_Results_64_bytes_1[2];
	PlcInputs._7600_Results_64_bytes_1[3] := HwInputs._7600_Results_64_bytes_1[3];
	PlcInputs._7600_Results_64_bytes_1[4] := HwInputs._7600_Results_64_bytes_1[4];
	PlcInputs._7600_Results_64_bytes_1[5] := HwInputs._7600_Results_64_bytes_1[5];
	PlcInputs._7600_Results_64_bytes_1[6] := HwInputs._7600_Results_64_bytes_1[6];
	PlcInputs._7600_Results_64_bytes_1[7] := HwInputs._7600_Results_64_bytes_1[7];
	PlcInputs._7600_Results_64_bytes_1[8] := HwInputs._7600_Results_64_bytes_1[8];
	PlcInputs._7600_Results_64_bytes_1[9] := HwInputs._7600_Results_64_bytes_1[9];
	PlcInputs._7600_Results_64_bytes_1[10] := HwInputs._7600_Results_64_bytes_1[10];
	PlcInputs._7600_Results_64_bytes_1[11] := HwInputs._7600_Results_64_bytes_1[11];
	PlcInputs._7600_Results_64_bytes_1[12] := HwInputs._7600_Results_64_bytes_1[12];
	PlcInputs._7600_Results_64_bytes_1[13] := HwInputs._7600_Results_64_bytes_1[13];
	PlcInputs._7600_Results_64_bytes_1[14] := HwInputs._7600_Results_64_bytes_1[14];
	PlcInputs._7600_Results_64_bytes_1[15] := HwInputs._7600_Results_64_bytes_1[15];
	PlcInputs._7600_Results_64_bytes_1[16] := HwInputs._7600_Results_64_bytes_1[16];
	PlcInputs._7600_Results_64_bytes_1[17] := HwInputs._7600_Results_64_bytes_1[17];
	PlcInputs._7600_Results_64_bytes_1[18] := HwInputs._7600_Results_64_bytes_1[18];
	PlcInputs._7600_Results_64_bytes_1[19] := HwInputs._7600_Results_64_bytes_1[19];
	PlcInputs._7600_Results_64_bytes_1[20] := HwInputs._7600_Results_64_bytes_1[20];
	PlcInputs._7600_Results_64_bytes_1[21] := HwInputs._7600_Results_64_bytes_1[21];
	PlcInputs._7600_Results_64_bytes_1[22] := HwInputs._7600_Results_64_bytes_1[22];
	PlcInputs._7600_Results_64_bytes_1[23] := HwInputs._7600_Results_64_bytes_1[23];
	PlcInputs._7600_Results_64_bytes_1[24] := HwInputs._7600_Results_64_bytes_1[24];
	PlcInputs._7600_Results_64_bytes_1[25] := HwInputs._7600_Results_64_bytes_1[25];
	PlcInputs._7600_Results_64_bytes_1[26] := HwInputs._7600_Results_64_bytes_1[26];
	PlcInputs._7600_Results_64_bytes_1[27] := HwInputs._7600_Results_64_bytes_1[27];
	PlcInputs._7600_Results_64_bytes_1[28] := HwInputs._7600_Results_64_bytes_1[28];
	PlcInputs._7600_Results_64_bytes_1[29] := HwInputs._7600_Results_64_bytes_1[29];
	PlcInputs._7600_Results_64_bytes_1[30] := HwInputs._7600_Results_64_bytes_1[30];
	PlcInputs._7600_Results_64_bytes_1[31] := HwInputs._7600_Results_64_bytes_1[31];
	PlcInputs._7600_Results_64_bytes_1[32] := HwInputs._7600_Results_64_bytes_1[32];
	PlcInputs._7600_Results_64_bytes_1[33] := HwInputs._7600_Results_64_bytes_1[33];
	PlcInputs._7600_Results_64_bytes_1[34] := HwInputs._7600_Results_64_bytes_1[34];
	PlcInputs._7600_Results_64_bytes_1[35] := HwInputs._7600_Results_64_bytes_1[35];
	PlcInputs._7600_Results_64_bytes_1[36] := HwInputs._7600_Results_64_bytes_1[36];
	PlcInputs._7600_Results_64_bytes_1[37] := HwInputs._7600_Results_64_bytes_1[37];
	PlcInputs._7600_Results_64_bytes_1[38] := HwInputs._7600_Results_64_bytes_1[38];
	PlcInputs._7600_Results_64_bytes_1[39] := HwInputs._7600_Results_64_bytes_1[39];
	PlcInputs._7600_Results_64_bytes_1[40] := HwInputs._7600_Results_64_bytes_1[40];
	PlcInputs._7600_Results_64_bytes_1[41] := HwInputs._7600_Results_64_bytes_1[41];
	PlcInputs._7600_Results_64_bytes_1[42] := HwInputs._7600_Results_64_bytes_1[42];
	PlcInputs._7600_Results_64_bytes_1[43] := HwInputs._7600_Results_64_bytes_1[43];
	PlcInputs._7600_Results_64_bytes_1[44] := HwInputs._7600_Results_64_bytes_1[44];
	PlcInputs._7600_Results_64_bytes_1[45] := HwInputs._7600_Results_64_bytes_1[45];
	PlcInputs._7600_Results_64_bytes_1[46] := HwInputs._7600_Results_64_bytes_1[46];
	PlcInputs._7600_Results_64_bytes_1[47] := HwInputs._7600_Results_64_bytes_1[47];
	PlcInputs._7600_Results_64_bytes_1[48] := HwInputs._7600_Results_64_bytes_1[48];
	PlcInputs._7600_Results_64_bytes_1[49] := HwInputs._7600_Results_64_bytes_1[49];
	PlcInputs._7600_Results_64_bytes_1[50] := HwInputs._7600_Results_64_bytes_1[50];
	PlcInputs._7600_Results_64_bytes_1[51] := HwInputs._7600_Results_64_bytes_1[51];
	PlcInputs._7600_Results_64_bytes_1[52] := HwInputs._7600_Results_64_bytes_1[52];
	PlcInputs._7600_Results_64_bytes_1[53] := HwInputs._7600_Results_64_bytes_1[53];
	PlcInputs._7600_Results_64_bytes_1[54] := HwInputs._7600_Results_64_bytes_1[54];
	PlcInputs._7600_Results_64_bytes_1[55] := HwInputs._7600_Results_64_bytes_1[55];
	PlcInputs._7600_Results_64_bytes_1[56] := HwInputs._7600_Results_64_bytes_1[56];
	PlcInputs._7600_Results_64_bytes_1[57] := HwInputs._7600_Results_64_bytes_1[57];
	PlcInputs._7600_Results_64_bytes_1[58] := HwInputs._7600_Results_64_bytes_1[58];
	PlcInputs._7600_Results_64_bytes_1[59] := HwInputs._7600_Results_64_bytes_1[59];
	PlcInputs._7600_Results_64_bytes_1[60] := HwInputs._7600_Results_64_bytes_1[60];
	PlcInputs._7600_Results_64_bytes_1[61] := HwInputs._7600_Results_64_bytes_1[61];
	PlcInputs._7600_Results_64_bytes_1[62] := HwInputs._7600_Results_64_bytes_1[62];
	PlcInputs._7600_Results_64_bytes_1[63] := HwInputs._7600_Results_64_bytes_1[63];
	PlcInputs._7600_Results_64_bytes_1[64] := HwInputs._7600_Results_64_bytes_1[64];
	PlcInputs._7600_Results_64_bytes_1[65] := HwInputs._7600_Results_64_bytes_1[65];
	PlcInputs._7600_Results_64_bytes_1[66] := HwInputs._7600_Results_64_bytes_1[66];
	PlcInputs._7600_Results_64_bytes_1[67] := HwInputs._7600_Results_64_bytes_1[67];
END_FUNCTION
